FUNCTION_BLOCK DataManager
VAR
	Settings : stSettings;
	{attribute addProperty Name "Save to database" }
	SaveSettings : CSharpMethod;
	{attribute clr [RenderIgnore()]}
	Invoke :BOOL;
END_VAR

IF Invoke THEN
	IF Save() THEN
		Invoke :=FALSE;	
	END_IF
END_IF

METHOD Save : BOOL
VAR_INPUT
END_VAR
Save := SaveSettings.Invoke();
END_METHOD

END_FUNCTION_BLOCK

(* stored: Version 1.1.0.1, ProductVersion 3.1.4024.5
   POU DataManager: Id {764204d4-1e96-47b0-8035-796674c2a74b}, SpecialFunc None
   Method Save: Id {74092171-1644-4089-9273-6edaf4d4fafa} *)
